FUNCTION_BLOCK FB_PTPArona EXTENDS FB_RecipeBase

METHOD Build : BOOL
VAR_INST
    TotalY          : REAL;
    TotalX          : REAL;
    ShorterY        : REAL;
    ShorterX        : REAL;
END_VAR
_Busy := TRUE;
_Done := FALSE;
_Error := FALSE;
Build := FALSE;
// 1. Zlecenie przeliczenia gabarytów, footrpintu i limitów klasie bazowej
THIS^.UpdateNestingLimits();

// 2. Jeśli detal wystaje poza maszynę - przerywamy od razu!
IF NOT _Config.IsValid THEN
    _Busy := FALSE;
    _Error := TRUE; 
    Build := FALSE;
    RETURN;
END_IF

// 3. Pobieramy wyliczone gabaryty nominalne do lokalnych zmiennych roboczych
TotalX   := _NominalX;
TotalY   := _NominalY; 

// ------------------------------------
// 1. Segregracja frezowania (Grooving)
// ------------------------------------
_SegmentsToGroove := 2;

_SegmentsGroove[1].Start.X := _Config.PanelHeight;
_SegmentsGroove[1].Stop.X  := _Config.PanelHeight;
_SegmentsGroove[1].Start.Y := TotalY;
_SegmentsGroove[1].Stop.Y  := 0;

_SegmentsGroove[2].Start.X :=  _Config.PanelHeight + 40;    
_SegmentsGroove[2].Stop.X  :=  _Config.PanelHeight + 40;    
_SegmentsGroove[2].Start.Y :=  TotalY;
_SegmentsGroove[2].Stop.Y  :=  0;                      


// ------------------------------------
// 2. Cięcie w osi X (Cut X)
// ------------------------------------+ 
_SegmentsToCutX := 2;

// Short Box Segments
_SegmentsCutX[1].Start.X := TotalX + _Config.CuttingOverpass;
_SegmentsCutX[1].Stop.X  := -_Config.CuttingOverpass;
_SegmentsCutX[1].Start.Y := 0;
_SegmentsCutX[1].Stop.Y  := 0;        

_SegmentsCutX[2].Start.X := TotalX + _Config.CuttingOverpass;                         
_SegmentsCutX[2].Stop.X  := - _Config.CuttingOverpass;                          
_SegmentsCutX[2].Start.Y := TotalY;
_SegmentsCutX[2].Stop.Y  := TotalY;        

// ------------------------------------
// 3. Cięcie w osi Y (Cut Y)
// ------------------------------------
_SegmentsToCutY := 2;

// Short Box Segments
_SegmentsCutY[1].Start.X := 0;                               
_SegmentsCutY[1].Stop.X  := 0;                               
_SegmentsCutY[1].Start.Y := TotalY +_Config.CuttingOverpass; 
_SegmentsCutY[1].Stop.Y  := -_Config.CuttingOverpass;        

_SegmentsCutY[2].Start.X := TotalX;                          
_SegmentsCutY[2].Stop.X  := TotalX;                          
_SegmentsCutY[2].Start.Y := TotalY +_Config.CuttingOverpass; 
_SegmentsCutY[2].Stop.Y  := -_Config.CuttingOverpass;        

_Busy := FALSE;
_Done := TRUE;
Build := TRUE;
END_METHOD

METHOD PROTECTED CalculateFootprint
VAR_INPUT
END_VAR
// BorgoWings wie, że jego wymiar powiększa się o ścianki zagięcia:
_NominalX := (2.0 * _Config.PanelHeight) + 40.0; 
_NominalY := _Config.PanelFrontLength;
END_METHOD

PROPERTY ExecutionRoute : E_ExecutionRoute
GET
ExecutionRoute := E_ExecutionRoute.ePTP;
END_GET
END_PROPERTY

METHOD FB_init : BOOL
VAR_INPUT
	bInitRetains : BOOL; // if TRUE, the retain variables are initialized (warm start / cold start)
	bInCopyCode : BOOL;  // if TRUE, the instance afterwards gets moved into the copy code (online change)
END_VAR
_Limits.PanelFrontLength.MinVal := 12.0;
_Limits.PanelFrontLength.MaxVal := 1234.0;

_Limits.PanelFrontWidth.MinVal  := 12.0;
_Limits.PanelFrontWidth.MaxVal  := 1234.0;

_Limits.PanelHeight.MinVal      := 12.0;
_Limits.PanelHeight.MaxVal      := 1234.0;

_Limits.RailHeightCorrection.MinVal := 12.0;
_Limits.RailHeightCorrection.MaxVal := 1234.0;

_Limits.CuttingOverpass.MinVal := 0.0;
_Limits.CuttingOverpass.MaxVal := 50.0;

_Limits.GroovingOverpass.MinVal := 0.0;
_Limits.GroovingOverpass.MaxVal := 50.0;

_Limits.GrooveDepthZ.MinVal := 0.0;
_Limits.GrooveDepthZ.MaxVal := 9.0; //
END_METHOD

END_FUNCTION_BLOCK

(* stored: Version 1.1.0.1, ProductVersion 3.1.4024.15
   POU FB_PTPArona: Id {a7865aba-34a9-4367-9b70-65119865d0af}, SpecialFunc None
   Method Build: Id {888409fe-0b8e-46d6-8abb-5ebdab25e661}
   Method CalculateFootprint: Id {330d8601-fd3b-4246-bed6-324b0a3cab48}
   Property ExecutionRoute: Id {7f69a90b-27cb-4780-8d18-f5335cbac906}
   Get Get: Id {c5f16da5-eee5-4f57-aa31-bf581754b3b8}
   Method FB_init: Id {fc78a4c1-f2de-4ec3-8288-cc1bf83cb800} *)
